FUNCTION_BLOCK RunUnitCellularC EXTENDS RunUnitTransporterBase
VAR_INPUT
END_VAR
VAR_OUTPUT
END_VAR
VAR
	//devices
	reachSensor : POINTER TO RunSignal;
	interfereSensor : POINTER TO RunSignal;
	holderCylinder : POINTER TO RunCylinder;
	pusherCylinder : POINTER TO RunCylinder;
	//liner
	liner : POINTER TO RunAxis;
	ptLinerSend : POINTER TO ParameterSet;
	ptLinerWork : POINTER TO ParameterSet;
	ptLinerReceive : POINTER TO ParameterSet;
	//rotator (option
	rotator : POINTER TO RunAxis;
	ptRotatorMutual : POINTER TO ParameterSet;
	ptRotatorSend : POINTER TO ParameterSet;
	ptRotatorReceive : POINTER TO ParameterSet;
END_VAR
VAR PERSISTENT
	//TODO memorize carrier existed?
END_VAR

SUPER^();
//inherits sync/mat relative variables

//interfere auto cut axis	(high priority


CASE outputState OF 
	eSpecialStates.INITIAL_BEGIN:
		IF rotator=0 or (rotator<>0 AND_THEN rotator^.ExecuteParameter(ptRotatorMutual)) THEN
			NextState := eSpecialStates.INITIAL_END;
		END_IF	
	//-----------------switch function
	0:
		IF reachSensor^.debouncedOn THEN
			//occupied , sending procedure
			NextState := 16#2000;
		ELSE
			//vacuumed , receiving procedure
			NextState := 16#1000;
		END_IF
	//-----------------sending procedure 
	16#2000:
		IF holderCylinder^.Execute(eCylinderCommands.COMMAND_B) AND NOT transitionByte.0 THEN
			transitionByte.0 := TRUE;
		END_IF
		IF pusherCylinder^.Execute(eCylinderCommands.COMMAND_A) AND NOT transitionByte.1 THEN
			transitionByte.1 := TRUE;
		END_IF
		IF transitionByte = 16#3 AND interfereSensor^.debouncedOff THEN
			bSerialTransition := TRUE;
		END_IF
	16#2001:
		bSerialTransition := rotator=0 OR (rotator<>0 AND_THEN rotator^.ExecuteParameter(ptRotatorMutual)); //otherwise would interfere
	16#2002:
		bSerialTransition := liner^.ExecuteParameter(ptLinerSend);
	16#2003:
		bSerialTransition := rotator=0 OR (rotator<>0 AND_THEN rotator^.ExecuteParameter(ptRotatorSend)); //reached then rotate
	16#2004:
		IF holderCylinder^.Execute(eCylinderCommands.COMMAND_A) THEN
			//release , wait to send
			syncEngaged := TRUE;
			bSerialTransition := TRUE;
		END_IF
	16#2005:
		IF syncAcknowledged AND_THEN pusherCylinder^.Execute(eCylinderCommands.COMMAND_B) THEN
			//go out
			bSerialTransition := TRUE;
		END_IF
	16#2006:
		IF interfereSensor^.debouncedOff AND reachSensor^.debouncedOff THEN
			syncEngaged := FALSE;//leaved
			bSerialTransition := TRUE;
		END_IF
	16#2007:
		IF pusherCylinder^.Execute(eCylinderCommands.COMMAND_A) AND NOT syncAcknowledged THEN
			//make sure synchronized
			NextState := 0; //rewind
		END_IF
	//---------------------receiving procedure
	16#1000:
		// holder off , pusher off , rotator/linear in receive position
		IF holderCylinder^.Execute(eCylinderCommands.COMMAND_A) AND NOT transitionByte.0 THEN
			transitionByte.0 := TRUE;
		END_IF
		IF pusherCylinder^.Execute(eCylinderCommands.COMMAND_A) AND NOT transitionByte.1 THEN
			transitionByte.1 := TRUE;
		END_IF
		IF (rotator=0 OR (rotator<>0 AND_THEN rotator^.ExecuteParameter(ptRotatorReceive))) AND NOT transitionByte.2 THEN
			transitionByte.2 := TRUE;
		END_IF
		IF liner^.ExecuteParameter(ptLinerReceive) AND not transitionByte.3 THEN
			transitionByte.3 := TRUE;
		END_IF
		IF transitionByte = 16#F AND interfereSensor^.debouncedOff THEN
			bSerialTransition := TRUE;
		END_IF
	16#1001:
		IF Upstream<>0 AND_THEN Upstream^.syncEngaged THEN
			Upstream^.syncAcknowledged := TRUE; //
			bSerialTransition := TRUE;
		END_IF
	16#1002:
		bSerialTransition := interfereSensor^.debouncedOff AND reachSensor^.debouncedOn;
	16#1003:
		IF Upstream<>0 AND_THEN NOT Upstream^.syncEngaged THEN
			Upstream^.syncAcknowledged := FALSE; //completely follow upstream ,
			bSerialTransition := TRUE;
		END_IF
	16#1004:
		IF holderCylinder^.Execute(eCylinderCommands.COMMAND_B) THEN
			NextState := 0;
		END_IF
END_CASE

METHOD FB_init : BOOL
VAR_INPUT
	bInitRetains : BOOL; // if TRUE, the retain variables are initialized (warm start / cold start)
	bInCopyCode : BOOL;  // if TRUE, the instance afterwards gets moved into the copy code (online change)
	
	argParent : POINTER TO RunUnitGeneric;
	argSlotBase : POINTER TO MaterialBlock;
	argSlotLast : POINTER TO MaterialBlock;
	
	argUpstream : POINTER TO RunUnitTransporterBase;
	
	argLinear : POINTER TO RunAxis;
	argRotator : POINTER TO RunAxis;
	argReachSensor : POINTER TO RunSignal;
	argInterfereSensor : POINTER TO RunSignal;
	argHolderCylinder : POINTER TO RunCylinder;
	argPusherCylinder : POINTER TO RunCylinder;
END_VAR
VAR CONSTANT
	indexSend : INT := 1;
	indexReceive : INT := 2;
	indexMutual : INT := 3; //equals to work position to Cellular D
END_VAR
//initialize 
Parent := argParent;
SlotBase := argSlotBase;
SlotLast := argSlotLast;

Upstream := argUpstream;

IF Upstream=0 THEN
	isProxyMode:=TRUE; //no upstream , i am proxy
END_IF

//device link
liner := argLinear;

reachSensor := argReachSensor;
interfereSensor := argInterfereSensor;
holderCylinder := argHolderCylinder;
pusherCylinder := argPusherCylinder;
//position link
ptLinerSend := ADR(liner^.ptpCommands[indexSend]);
ptLinerReceive := ADR(liner^.ptpCommands[indexReceive]);
ptLinerWork := ADR(liner^.ptpCommands[indexMutual]);
// rotator(option
IF argRotator <> 0 THEN
	rotator := argRotator;
	
	ptRotatorSend := ADR(rotator^.ptpCommands[indexSend]);
	ptRotatorReceive := ADR(rotator^.ptpCommands[indexReceive]);
	ptRotatorMutual := ADR(rotator^.ptpCommands[indexMutual]);
END_IF
END_METHOD

END_FUNCTION_BLOCK

(* stored: Version 1.1.0.1, ProductVersion 3.1.4022.10
   POU RunUnitCellularC: Id {0b9fe5c8-2bef-4f04-b3ac-e69748226c8f}, SpecialFunc None
   Method FB_init: Id {a9a51c1b-f758-4ded-9a6c-01bf50e17b39} *)
